// TIA Portal V20 export
ORGANIZATION_BLOCK "Startup"   // OB1000, LAD, Startup
TITLE = "Complete Restart"
// This block is called only once in the very first PLC cycle after STOP -> RUN.
// Configuration seetings and assignemts are to be programmed here.
// stored: AutoNumber false, IsIECCheckEnabled true, Namespace Unit1, SetENOAutomatically true
   VAR_INPUT
      LostRetentive : Bool;   // True if retentive data are lost
      LostRTC : Bool;   // True if date and time are lost
   END_VAR
   VAR_TEMP
      tempIndex : Int;   // Index of Unit in the array
   END_VAR
BEGIN

REGION Network 1: Unit Index Number
   // Assign the number of the unit to a temp for correct array index access.
   // Number is defined in PLC tags of Software Unit Global.
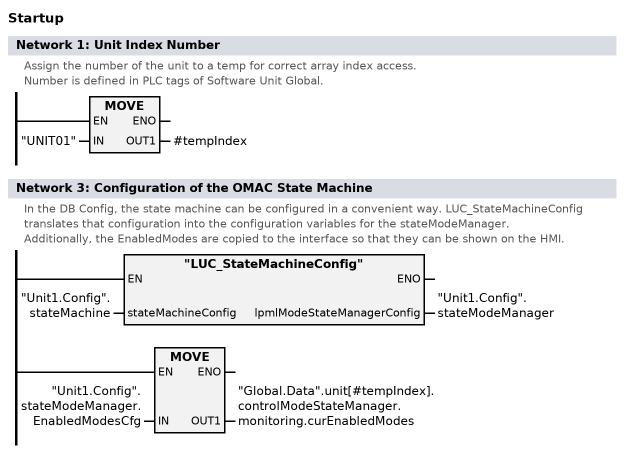
   RUNG wire#powerrail
      Move(in := "UNIT01", out1 => #tempIndex)
   END_RUNG
   // the same network as SCL:
   #tempIndex := "UNIT01";
END_REGION

REGION Network 2 (SCL): Build the Absolut Reference Designator
   // Set the Absoult Reference Designator in the DB Config. It is combined out of the parent reference designator and the own reference designator (=relative)
   IF LEN(IN := "Unit1.Config".unit.referenceDesignator.parent) <> 0 THEN
       "Unit1.Config".unit.referenceDesignator.combined := CONCAT_WSTRING(IN1 := "Unit1.Config".unit.referenceDesignator.parent, IN2 := WSTRING#'.', IN3 := "Unit1.Config".unit.referenceDesignator.relative);
   ELSE
       "Unit1.Config".unit.referenceDesignator.combined := "Unit1.Config".unit.referenceDesignator.relative;
   END_IF;
END_REGION

REGION Network 3: Configuration of the OMAC State Machine
   // In the DB Config, the state machine can be configured in a convenient way. LUC_StateMachineConfig translates that configuration into the configuration variables for the stateModeManager.
   // Additionally, the EnabledModes are copied to the interface so that they can be shown on the HMI.
   RUNG wire#powerrail
      "LUC_StateMachineConfig"(stateMachineConfig := "Unit1.Config".stateMachine, lpmlModeStateManagerConfig => "Unit1.Config".stateModeManager)
   END_RUNG
   RUNG wire#powerrail
      Move(in := "Unit1.Config".stateModeManager.EnabledModesCfg, out1 => "Global.Data".unit[#tempIndex].controlModeStateManager.monitoring.curEnabledModes)
   END_RUNG
   // the same network as SCL:
   "LUC_StateMachineConfig"(stateMachineConfig := "Unit1.Config".stateMachine,
                           lpmlModeStateManagerConfig => "Unit1.Config".stateModeManager);
   "Global.Data".unit[#tempIndex].controlModeStateManager.monitoring.curEnabledModes := "Unit1.Config".stateModeManager.EnabledModesCfg;
END_REGION

REGION Network 4 (SCL): Startup
   // SLM
   "Unit1.Config".SLM := "BA010AZCRCU1~BA010AZCRCU1_X150~S220_SLM_36_108_kW_SIEMENS_,,,";

   // BA30
   "Unit1.Config".BA030.SEND.connectionId := 16#0112;
   "Unit1.Config".BA030.SEND.rid := 16#0000_0012;
   "Unit1.Config".BA030.RCV.connectionId := 16#0112;
   "Unit1.Config".BA030.RCV.rid := 16#0000_0011;

   // BA40
   "Unit1.Config".BA040.SEND.connectionId := 16#0122;
   "Unit1.Config".BA040.SEND.rid := 16#0000_0022;
   "Unit1.Config".BA040.RCV.connectionId := 16#0122;
   "Unit1.Config".BA040.RCV.rid := 16#0000_0021;

   // FFU
   "Unit1.Config".cmFFU.MB_Comm_Load.PORT := 732;
   "Unit1.Config".cmFFU.MB_Comm_Load.BAUD := 9600;
END_REGION
END_ORGANIZATION_BLOCK
